// TIA Portal V16 export
// export: Created 2019-09-22T13:34:01.4059862Z, ExportSetting WithDefaults, DisplayName Totally Integrated Automation Portal, DisplayVersion V16, DisplayName TIA Portal Version Control Interface, DisplayVersion V16, DisplayName TIA Portal Openness, DisplayVersion V16, DisplayName STEP 7 Professional, DisplayVersion V16, DisplayName SIMATIC Energy Suite, DisplayVersion V16, DisplayName STEP 7 Safety, DisplayVersion V16, DisplayName WinCC Professional, DisplayVersion V16, DisplayName SIMATIC Visualization Architect, DisplayVersion V16
FUNCTION_BLOCK "LiftCmd"   // FB190, LAD
{ S7_Optimized_Access := 'TRUE' }
VERSION : 0.1
// stored: AutoNumber true, IsIECCheckEnabled false, IsRetainMemResEnabled false, MemoryReserve 100, SetENOAutomatically false, UDAEnableTagReadback false
   VAR_INPUT
      interLockAuto : Bool;   // Interlock automatic
      interLockMan : Bool;   // Interlock manual
      autoStarted : Bool;   // Automatic started
      startLiftUp : Bool;   // Start lift up
      startLiftDown : Bool;   // Start lift down
      manLiftUp : Bool;   // Manual start lift up
      manLiftDown : Bool;   // Manual start lift down
      sensorLiftUp : Bool;   // Sensor lift up
      sensorLiftDown : Bool;   // Sensor lift down
   END_VAR
   VAR_OUTPUT
      outLiftUp : Bool;   // Output lift up
      outLiftDown : Bool;   // Output lift down
   END_VAR
   VAR
      statTrigLiftUp : Bool;   // Trigger lift up
      statTrigLiftDown : Bool;   // Trigger lift down
   END_VAR
   VAR_TEMP
      tempUnLock : Bool;
   END_VAR
BEGIN

REGION Network 1: set trigger lift up
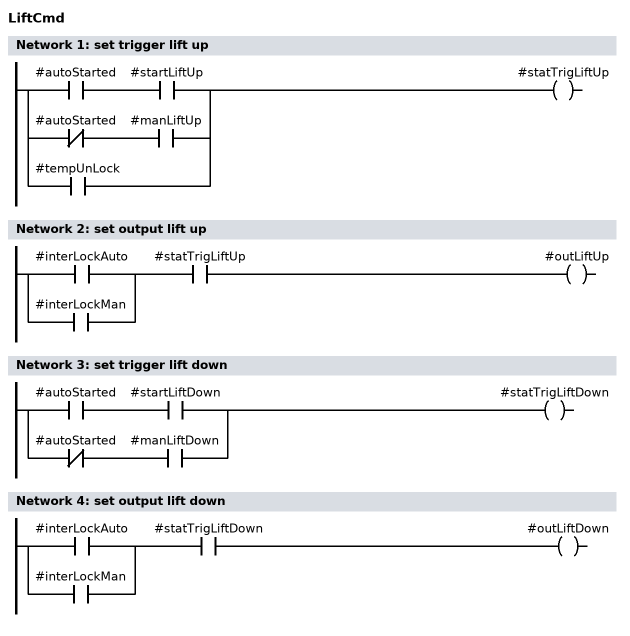
   RUNG wire#powerrail
      Contact( #autoStarted )
      Contact( #startLiftUp )
      wire#w1
      Coil( #statTrigLiftUp )
   END_RUNG
   RUNG wire#powerrail
      I_Contact( #autoStarted )
      Contact( #manLiftUp )
   END_RUNG wire#w1
   RUNG wire#powerrail
      Contact( #tempUnLock )
   END_RUNG wire#w1
   // the same network as SCL:
   #statTrigLiftUp := (#autoStarted AND #startLiftUp) OR (NOT #autoStarted AND #manLiftUp) OR #tempUnLock;
END_REGION

REGION Network 2: set output lift up
   RUNG wire#powerrail
      Contact( #interLockAuto )
      wire#w1
      Contact( #statTrigLiftUp )
      Coil( #outLiftUp )
   END_RUNG
   RUNG wire#powerrail
      Contact( #interLockMan )
   END_RUNG wire#w1
   // the same network as SCL:
   #outLiftUp := (#interLockAuto OR #interLockMan) AND #statTrigLiftUp;
END_REGION

REGION Network 3: set trigger lift down
   RUNG wire#powerrail
      Contact( #autoStarted )
      Contact( #startLiftDown )
      wire#w1
      Coil( #statTrigLiftDown )
   END_RUNG
   RUNG wire#powerrail
      I_Contact( #autoStarted )
      Contact( #manLiftDown )
   END_RUNG wire#w1
   // the same network as SCL:
   #statTrigLiftDown := (#autoStarted AND #startLiftDown) OR (NOT #autoStarted AND #manLiftDown);
END_REGION

REGION Network 4: set output lift down
   RUNG wire#powerrail
      Contact( #interLockAuto )
      wire#w1
      Contact( #statTrigLiftDown )
      Coil( #outLiftDown )
   END_RUNG
   RUNG wire#powerrail
      Contact( #interLockMan )
   END_RUNG wire#w1
   // the same network as SCL:
   #outLiftDown := (#interLockAuto OR #interLockMan) AND #statTrigLiftDown;
END_REGION
END_FUNCTION_BLOCK
